(* PLC project Sin nombre, Desconocido Sin nombre 1 *)
(* stored: creationDateTime 2022-11-03T18:46:07, modificationDateTime 2022-11-07T02:13:38 *)

PROGRAM program0
  VAR
    OUT AT %QX0.0 : BOOL := 0;
    OUT0 AT %QX0.1 : BOOL := 0;
    OUT1 AT %QX0.2 : BOOL := 0;
    OUT2 AT %QX0.3 : BOOL := 0;
    IN AT %IX0.0 : BOOL := 0;
  END_VAR
  VAR
    TP0 : TP;
    TOF0 : TOF;
    CTU0 : CTU;
    delay : TIME;
  END_VAR
  VAR  (* added by the conversion: wires and edge detectors of the diagram *)
    R_TRIG1 : R_TRIG;
    _EQ21_OUT : BOOL;
    _EQ11_OUT : BOOL;
    _EQ27_OUT : BOOL;
    _EQ20_OUT : BOOL;
  END_VAR

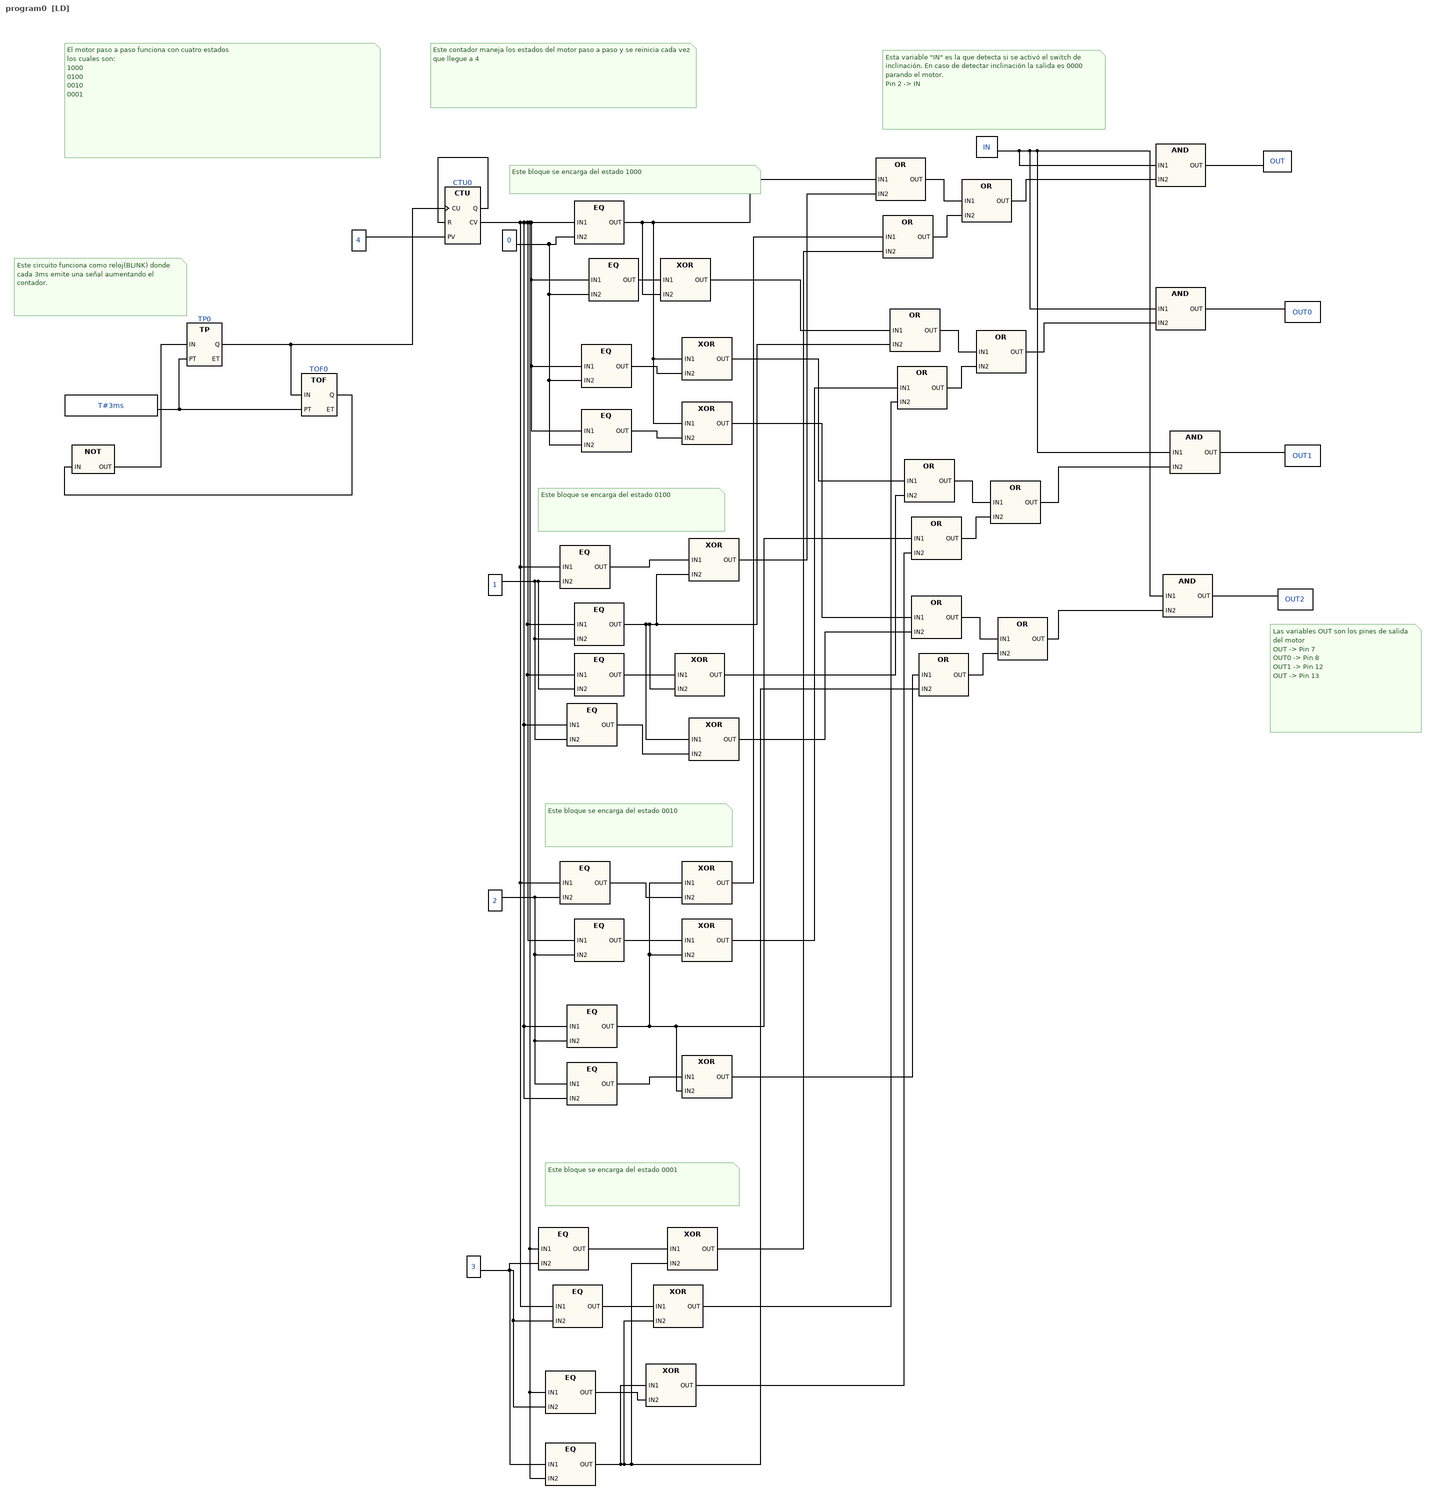
(* LD diagram, written out as Structured Text *)
(* El motor paso a paso funciona con cuatro estados
los cuales son:
1000
0100
0010
0001 *)
(* Este contador maneja los estados del motor paso a paso y se reinicia cada vez que llegue a 4 *)
(* Esta variable "IN" es la que detecta si se activó el switch de inclinación. En caso de detectar inclinación la salida es 0000 parando el motor.
Pin 2 -> IN *)
TOF0(IN := TP0.Q, PT := T#3ms);
TP0(IN := NOT TOF0.Q, PT := T#3ms);
R_TRIG1(CLK := TP0.Q);
CTU0(CU := R_TRIG1.Q, R := CTU0.Q, PV := 4);
_EQ21_OUT := CTU0.CV = 0;
_EQ11_OUT := CTU0.CV = 1;
_EQ27_OUT := CTU0.CV = 2;
_EQ20_OUT := 3 = CTU0.CV;
OUT := IN AND (_EQ21_OUT OR CTU0.CV = 1 XOR _EQ11_OUT OR _EQ27_OUT XOR CTU0.CV = 2 OR CTU0.CV = 3 XOR _EQ20_OUT);
(* Este bloque se encarga del estado 1000 *)
(* Este circuito funciona como reloj(BLINK) donde cada 3ms emite una señal aumentando el contador. *)
OUT0 := IN AND (CTU0.CV = 0 XOR _EQ21_OUT OR _EQ11_OUT OR CTU0.CV = 2 XOR _EQ27_OUT OR CTU0.CV = 3 XOR _EQ20_OUT);
OUT1 := IN AND (_EQ21_OUT XOR CTU0.CV = 0 OR CTU0.CV = 1 XOR _EQ11_OUT OR _EQ27_OUT OR _EQ20_OUT XOR CTU0.CV = 3);
(* Este bloque se encarga del estado 0100 *)
OUT2 := IN AND (_EQ21_OUT XOR CTU0.CV = 0 OR _EQ11_OUT XOR CTU0.CV = 1 OR 2 = CTU0.CV XOR _EQ27_OUT OR _EQ20_OUT);
(* Las variables OUT son los pines de salida del motor
OUT -> Pin 7
OUT0 -> Pin 8
OUT1 -> Pin 12
OUT -> Pin 13 *)
(* Este bloque se encarga del estado 0010 *)
(* Este bloque se encarga del estado 0001 *)
END_PROGRAM

CONFIGURATION Config0
  RESOURCE Res0 ON PLC
    TASK task0(INTERVAL := T#20ms, PRIORITY := 0);
    PROGRAM instance0 WITH task0 : program0;
  END_RESOURCE
END_CONFIGURATION
